// TIA Portal V18 export
VAR_GLOBAL   // PLC tag table "S2_R2"
   S2_R2_Valve_Up AT %Q600.0 : Bool;
   S2_R2_Valve_Down AT %Q600.1 : Bool;
   S2_R2_Sen_Drv_1 AT %Q600.2 : Bool;
   S2_R2_Sen_Drv_2 AT %Q600.3 : Bool;
   S2_R2_Sen_Drv_3 AT %Q600.4 : Bool;
   S2_R2_Sen_Drv_4 AT %Q600.5 : Bool;
   S2_R2_Sen_Val1_Up AT %Q600.6 : Bool;
   S2_R2_Sen_Val1_Down AT %Q600.7 : Bool;
   S2_R2_Sen_Val2_Up AT %Q601.0 : Bool;
   S2_R2_Sen_Val2_Down AT %Q601.1 : Bool;
   S2_R2_Hyd_Filtr AT %Q601.2 : Bool;
   S2_R2_Hyd_Empty AT %Q601.3 : Bool;
   S2_R2_Safety1_1 AT %I650.0 : Bool;
   S2_R2_Safety2_1 AT %I650.1 : Bool;
   S2_R2_Safety3_1 AT %I650.2 : Bool;
   S2_R2_Safety4_1 AT %I650.3 : Bool;
   S2_R2_Safety1_2 AT %I650.4 : Bool;
   S2_R2_Safety2_2 AT %I650.5 : Bool;
   S2_R2_Safety3_2 AT %I650.6 : Bool;
   S2_R2_Safety4_2 AT %I650.7 : Bool;
END_VAR
